FUNCTION_BLOCK FB_TestHTTP_Mindsphere_CreateMapping
VAR_INPUT
	bSend				: BOOL;
END_VAR
VAR_IN_OUT
	fbClient			: FB_IotHttpClient;
END_VAR
VAR_OUTPUT
	bBusy				: BOOL;
	bError				: BOOL;
END_VAR
VAR	
	fbRequest			: FB_IotHttpRequest;
	fbHeader			: FB_IotHttpHeaderFieldMap;
	fbJson				: FB_JsonDomParser;
	nState				: UDINT;
	RisingEdge			: R_TRIG;
	
	bGetContentResult	: BOOL;
	sContent			: STRING(2048);
	
	bGetJsonResult		: BOOL;
	jsonDoc				: SJsonValue;
	jsonVal				: SJsonValue;
	sResultValue		: STRING;
	
	nReqCount			: UDINT;
	nResCount			: UDINT;
	nValidResCount		: UDINT;
	nErrCount			: UDINT;	
END_VAR

RisingEdge(CLK:= bSend);
CASE nState OF
0:		
	IF RisingEdge.Q THEN
		// Body includes JSON document with DataSource configuration that should be created
		sContent := '{"agentId":"956cce3605b1420890095e50e2b11e17","dataPointId":"DP001_temprature_KLR","entityId":"956cce3605b1420890095e50e2b11e17","propertySetName":"SvenG_NB05_Aspect","propertyName":"Pump1"}';
		fbHeader.AddField('Content-Type', 'application/json', FALSE);
		// Header field 'Authorization' now includes RAT 
		fbHeader.AddField('Authorization', 'Bearer eyJraWQiOiJrZXktaWQtMSIsImFsZyI6IlJTMjU2IiwidHlwIjoiSldUIn0.eyJqdGkiOiJlY2I4Y2RkZS1jOTFhLTRkNGMtODA2Mi1lYTBmN2Y5ZGZkMjkiLCJzY29wZSI6WyJtZHNwOmNvcmU6RGVmYXVsdEFnZW50Il0sImlzcyI6Imh0dHBzOi8vc291dGhnYXRlLmV1MS5taW5kc3BoZXJlLmlvL2FwaS9hZ2VudG1hbmFnZW1lbnQvIiwic3ViIjoiOTU2Y2NlMzYwNWIxNDIwODkwMDk1ZTUwZTJiMTFlMTciLCJ6aWQiOiJhZ2VudGlhbSIsImF1ZCI6WyJzb3V0aGdhdGUiXSwiaWF0IjoxNTgyMTg4OTIwLCJleHAiOjE1ODIxOTI1MjAsInNjaGVtYXMiOlsidXJuOnNpZW1lbnM6bWluZHNwaGVyZTppYW06djEiXSwidGVuIjoiYmVja2hvZmYiLCJ0ZW5fY3R4IjoibWFpbi10ZW5hbnQiLCJjYXQiOiJhZ2VudC10b2tlbjp2MSIsImdyYW50X3R5cGUiOiJjbGllbnRfY3JlZGVudGlhbHMifQ.XLMR7pQDBiRZeDwtBLfKujJrPIWwvFw28DjtedfYL_x4iOUIcV7U6AJyKe6Wnit4GOAKfJYh_BGD160E3ns7RjRBYSx8Lj5dxI20l3g_KMcpgILoaW8gYlx41Y4q6W44zctJ04TQLsaz-Vc3eOEJ_TdMTGc_7s4v4YsQbZinKN-ZmQF_sXdGbihL2CkbqhnaubwZGn_FmSZosuiDXk4GFdF1TX2xXHQCz39p8jPYtgq2x9LkuIFtEzUct_lTy30rcwS2Fq6m-ac6gldJFtvqLZoXu3wUlHR1F7kAYndm6wvtXXlgDo5otTMZfzXBTEQA3JS2Cucys3gJNhYEDpUAtg', FALSE);
		IF fbRequest.SendRequest(sUri:= '/api/mindconnect/v3/dataPointMappings', fbClient:= fbClient, eRequestType:= ETcIotHttpRequestType.HTTP_POST, pContent:= ADR(sContent), nContentSize:= LEN2(ADR(sContent)), fbHeader:= fbHeader) THEN				
			nState:= 1;
			nReqCount:= nReqCount+1;
			bBusy:= TRUE;
			bError:= FALSE;
		END_IF					
	END_IF
1:
	IF NOT fbRequest.bBusy THEN
		bError:= TRUE;
		IF NOT fbRequest.bError THEN				 				
			bGetContentResult:= fbRequest.GetContent(pContent:= ADR(sContent), nContentSize:= SIZEOF(sContent), bSetNullTermination:= TRUE);	
			IF fbRequest.nStatusCode >= 200 AND fbRequest.nStatusCode < 300 THEN
				bGetJsonResult:= FALSE;
				jsonDoc:= fbRequest.GetJsonDomContent(fbJson);				
				(* Parse response in order to acquire created DatsSource configuration *)
				nResCount:= nResCount+1;					
			END_IF				
		END_IF
		nState:= 0;
		bBusy:= FALSE;
		IF bError THEN
			nErrCount:= nErrCount+1;
		END_IF		
	END_IF  	
END_CASE

END_FUNCTION_BLOCK

(* stored: Version 1.1.0.1, ProductVersion 3.1.4024.3
   POU FB_TestHTTP_Mindsphere_CreateMapping: Id {410f4342-2baf-4d27-b956-9cc1af0fdb5e}, SpecialFunc None *)
